(* PLC project model, Beckhoff Automation Beckhoff MLlib 3.1.251201.0 *)
(* stored: creationDateTime 2026-07-10T12:15:28.0358724, modificationDateTime 2026-07-10T12:15:28.0358724 *)

TYPE ST_modelInput :
STRUCT

	{attribute 'hide'} _header_DO_NOT_CHANGE : ARRAY[0..63] OF SINT := [-1,-112,120,86,52,18,-1,-1,1,-1,0,0,-1,-1,-112,-112,55,-22,8,-62,15,-11,-53,-120,-65,-26,40,-59,-103,80,20,5,37,-41,0,-16,-125,-33,-67,117,-59,70,-31,-53,-46,-33,-68,-19,80,2,0,0,0,0,0,0,0,0,0,0,0,0,0,0];
	in_input_tensor : ARRAY[0..0,0..32,0..3] OF REAL;

END_STRUCT
END_TYPE

TYPE ST_modelOutput :
STRUCT

	{attribute 'hide'} _header_DO_NOT_CHANGE : ARRAY[0..63] OF SINT := [-1,-112,120,86,52,18,-1,-1,1,-1,0,0,-1,-1,-112,-112,-35,24,-50,75,-65,96,-121,123,127,87,61,127,-39,-108,16,-70,120,-89,-28,78,-43,26,-32,-7,81,19,29,-89,-55,3,43,2,68,0,0,0,0,0,0,0,0,0,0,0,0,0,0,0];
	out_prediction_tensor : ARRAY[0..0,0..0] OF REAL;

END_STRUCT
END_TYPE
